(* IEC 61131-3 sources: SRCI/RobotLibrary/RobotLibrary/POUs/Read/MC_ReadActualTCPVelocity, 1 file *)

(* ---- MC_ReadActualTCPVelocityFB.st ---- *)
/// Read actual TCP velocity
FUNCTION_BLOCK MC_ReadActualTCPVelocityFB EXTENDS RobotLibraryBaseExecuteFB
// -------------------------------------------------------------------------
//  SRCI Robot Library
// -------------------------------------------------------------------------
//
//  Object:      ReadActualTCPVelocityFB
//  Author:      Thorsten Brach
//  Date:        2024-06-01
//
//  Description:
//
//
//  Copyright:
//    (C) 2024 Thorsten Brach. All rights reserved
//             Licensed under the LGPL-3.0 license.
//
//  Disclaimer:
//    This project is provided without any guarantee and can be used for
//    private and commercial purposes. Any use is at the user’s
//    own risk and responsibility.
//
// -------------------------------------------------------------------------
VAR_INPUT
  /// Processing mode
  ProcessingMode     : ProcessingMode;
  /// Defines the target sequence in which the command will be executed
  ///  For more information about the differentiation of sequences see chapter 5.5.3.4
  SequenceFlag       : SequenceFlag;
  /// command parameter
  ParCmd             : ReadActualTCPVelocityParCmd;
END_VAR

VAR_OUTPUT
  /// TRUE, while the following outputs return valid values:
  /// • ActualTCPVelocity
  /// • ToolNoReturn
  /// • FrameNoReturn
  Valid              : BOOL;
  /// The command was aborted by another command.
  CommandAborted     : BOOL;
  /// Command is transferred and confirmed by the RC
  CommandBuffered    : BOOL;
  /// TRUE, while command is interrupted during execution and can be continued
  CommandInterrupted : BOOL;
  /// Receiving of input parameter values has been acknowledged by RC
  ParameterAccepted  : BOOL;
  /// command outputs
  OutCmd             : ReadActualTCPVelocityOutCmd;
END_VAR

VAR
  /// internal copy of command parameter
 _parCmd             : ReadActualTCPVelocityParCmd;
  /// command data to send
 _command            : ReadActualTCPVelocitySendData;
  /// response data received
 _response           : ReadActualTCPVelocityRecvData;
END_VAR

  SUPER^(AxesGroup := AxesGroup);

END_FUNCTION_BLOCK

METHOD CheckParameterChanged : BOOL
VAR_IN_OUT
  /// Robot assignment of function
  AxesGroup    : AxesGroup;
END_VAR

  // Check ParCmd Size is > 0, becaue MemCmp does not work correctly with size = 0
  IF (SIZEOF(ParCmd) = 0)
  THEN
    RETURN;
  END_IF

  // compare memory
  CheckParameterChanged := ( MemCmp(ADR(ParCmd), ADR(_parCmd), SIZEOF(ParCmd)) <> RobotLibraryConstants.OK );

  IF ( CheckParameterChanged )
  THEN
    // update internal copy of parameters
   _parCmd := ParCmd;
    // inc parameter sequence
   _command.ParSeq := _command.ParSeq + 1;
    // update command data
    CommandData := CreateCommandPayload(); // ( Access via reference to rCommandFB in ACR )
    // notify active command register
    AxesGroup.Acyclic.ActiveCommandRegister.NotifyParameterChanged := _uniqueID;
    // Reset parameter accepted flag
    ParameterAccepted := FALSE;
  END_IF

END_METHOD

METHOD INTERNAL CreateCommandPayload : SendData
// Table 6-63: Sent CMD payload (PLC to RC) of "ReadActualTCPVelocity"
// --------------------------
// Header
// --------------------------
// Byte 00 : UINT  - Type HB
// Byte 01 :       - Type LB
// Byte 02 : USINT - Reserve | ExecutionMode
// Byte 03 : USINT - ParSeq  | Priority
// --------------------------
// Datablock
// --------------------------
// Byte 04 : USINT - ToolNo
// Byte 05 : USINT - FrameNo
// --------------------------

  // set command parameter
  _command.CmdTyp                    :=  CmdType.ReadActualTCPVelocity;
  _command.ExecMode                  :=  ExecMode;
  _command.ParSeq                    := _command.ParSeq;
  _command.Priority                  :=  Priority;
  _command.ToolNo                    := _parCmd.ToolNo;
  _command.FrameNo                   := _parCmd.FrameNo;

  // copy command data to header
  _cmdHeader := _command;
  // call base implementation to copy header to payload buffer
  CreateCommandPayload := SUPER^.CreateCommandPayload();

  // add command.ToolNo
  CreateCommandPayload.AddUsint(_command.ToolNo);
  // add command.FrameNo
  CreateCommandPayload.AddUsint(_command.FrameNo);

END_METHOD

METHOD FB_init : BOOL
VAR_INPUT
  /// if TRUE, the retain variables are initialized (warm start / cold start)
	bInitRetains : BOOL;
  /// if TRUE, the instance afterwards gets moved into the copy code (online change)
	bInCopyCode  : BOOL;
END_VAR

  MyType := 'MC_ReadActualTCPVelocityFB';

  ExecMode := ExecutionMode.PARALLEL;

END_METHOD

METHOD PROTECTED OnCall
VAR_IN_OUT
  /// Robot assignment of function
  AxesGroup : AxesGroup;
END_VAR

  // call base implementation
  SUPER^.OnCall(AxesGroup := AxesGroup);

  CASE _stepCmd OF

    00:  IF ( _execute_R.Q )
         THEN
           // set busy flag
           Busy := TRUE;
           // Reset command outputs
           MemSet(ADR(OutCmd),0,SIZEOF(OutCmd));
           // apply command parameter
          _parCmd := ParCmd;
           // init parameter sequence
          _command.ParSeq := 1;
           // set timeout
           SetTimeout(PT := _timeoutCmd, rTimer := _timerCmd);
           // inc step counter
          _stepCmd := _stepCmd + 1;
  	     END_IF

    01:  // create command data
         CommandData := CreateCommandPayload();
         // Add command to active command register
        _uniqueID := AxesGroup.Acyclic.ActiveCommandRegister.AddCmd( pCommandFB := ADR(THIS^ ));
         // set timeout
         SetTimeout(PT := _timeoutCmd, rTimer := _timerCmd);
         // inc step counter
        _stepCmd := _stepCmd + 1;

    02:  // Wait for responce received
         IF ( _responseReceived )
         THEN
           // reset response received flag
          _responseReceived := FALSE;

           CASE  _response.State
           OF
             CmdMessageState.BUFFERED    : CommandBuffered    := TRUE;
             CmdMessageState.ACTIVE      : ParameterAccepted  := TRUE;
             CmdMessageState.INTERRUPTED : CommandInterrupted := TRUE;
             CmdMessageState.DONE        : Done               := TRUE;
             CmdMessageState.ABORTED     : CommandAborted     := TRUE;
             CmdMessageState.ERROR       : Error              := TRUE;
  				 END_CASE

           // Done, Aborted or Error ?
           IF (_response.State >= CmdMessageState.DONE )
           THEN
             // Reset Busy flag
             Busy := FALSE;
             // Update results
             OutCmd.ToolNoReturn      := _response.ToolNoReturn;
             OutCmd.FrameNoReturn     := _response.FrameNoReturn;
             OutCmd.ActualTCPVelocity := _response.ActualTCPVelocity;

             // set timeout
             SetTimeout(PT := _timeoutCmd, rTimer := _timerCmd);
             // inc step counter
            _stepCmd := _stepCmd + 1;
  				 END_IF
         END_IF

    03: IF ( NOT Execute)
        THEN
          Reset();
  			END_IF
  ELSE
    // invalid step
    ErrorID := RobotLibraryEvents.ERR_INVALID_STEP;
  END_CASE

  // Cancel
  IF (Busy) AND (NOT Execute)
  THEN
    // try to remove cmd
    AxesGroup.Acyclic.ActiveCommandRegister.RemoveCmd(_uniqueID);
  END_IF

  // Reset FB
  IF ( NOT Execute )
  THEN
    Reset();
  END_IF

END_METHOD

METHOD INTERNAL ParseResponsePayload : DINT
// Table 6-64: Received CMD payload (RC to PLC) of " ReadActualTCPVelocity "
// --------------------------
// Header
// --------------------------
// Byte 00 : USINT   - ParSeq | State
// Byte 01 : SINT    - AlarmMessageSeverity
// Byte 02 : UINT    - AlarmMessageCode HB
// Byte 03 :         - AlarmMessageCode LB
// --------------------------
// Datablock
// --------------------------
// Byte 04 : USINT   - ToolNoReturn
// Byte 05 : USINT   - FrameNoReturn
// Byte 06 : REAL    - ActualTCPVelocity HW HB
// Byte 07 :           ActualTCPVelocity HW LB
// Byte 08 :           ActualTCPVelocity LW HB
// Byte 09 :           ActualTCPVelocity LW LB
// --------------------------
VAR_INPUT
  /// Response data
  ResponseData : RecvData;
END_VAR

  // call base implementation to parse the header from payload buffer
  ResponseData.PayloadPtr := SUPER^.ParseResponsePayload(ResponseData);

  // copy parsed header to response
  _response.ParSeq               := _rspHeader.ParSeq;
  _response.State                := _rspHeader.State;
  _response.AlarmMessageSeverity := _rspHeader.AlarmMessageSeverity;
  _response.AlarmMessageCode     := _rspHeader.AlarmMessageCode;

  // Get Response.ToolNoReturn
  _response.ToolNoReturn := ResponseData.GetUsint();
  // Get Response.FrameNoReturn
  _response.FrameNoReturn := ResponseData.GetUsint();
  // Get Response.ActualTCPVelocity
  _response.ActualTCPVelocity := ResponseData.GetReal();

END_METHOD

METHOD PROTECTED Reset : DINT
VAR_INPUT
END_VAR

  Reset := SUPER^.Reset();

  Done               := FALSE;
  Busy               := FALSE;
  Valid              := FALSE;
  ParameterAccepted  := FALSE;
  CommandBuffered    := FALSE;
  CommandAborted     := FALSE;
  CommandInterrupted := FALSE;

END_METHOD
